(* PLC project v0.6.04_CycleSemiAuto.project, CODESYS CODESYS V3.5 SP19 Patch 1 *)
(* stored: creationDateTime 2026-08-15T14:41:18.168777, modificationDateTime 2026-08-15T14:41:18.168777 *)

(* values of E_Mode: DISABLE: Mode Désactivé / Veille de sécurité (sorties bloquées); MAINT_N1: Manuel Niveau 1 : Pilotage unitaire avec toutes sécurités actives; MAINT_N2: Manuel Niveau 2 : Pilotage dégradé (droits étendus + bypasses autorisés); SEMI_AUTO: Mode Semi-Automatique (séquenceur automatique) *)

{attribute 'qualified_only'}
{attribute 'strict'}
TYPE E_Mode : (DISABLE := 0, MAINT_N1 := 1, MAINT_N2 := 2, SEMI_AUTO := 3);
END_TYPE

(* ═══════════════════════════════════════════════════════════════ 📡 ST_Diag_Device — Structure diagnostic d'un esclave ou bus ═══════════════════════════════════════════════════════════════ *)
TYPE ST_Diag_Device : STRUCT
  Online : BOOL;  (* Esclave visible sur le bus *)
  Operational : BOOL;  (* Esclave en mode OP (opérationnel) *)
  Error : BOOL;  (* Signal de défaut actif pour cet esclave *)
  ErrorId : WORD;  (* Code défaut détaillé *)
  State : E_Diag_State;  (* Phase courante du cycle de diagnostic *)
  StateAtError : E_Diag_State;  (* Instantané de la phase lors de l'anomalie *)
END_STRUCT;
END_TYPE

(* ═══════════════════════════════════════════════════════════════ 🕹️ ST_Joystick_AxisCmd — Consigne d'axe normalisée (sortie FB_Joystick) ─────────────────────────────────────────────────────────────── 📄 Doc métier : DOC/AF/AF_Partie-08_Fonction_Joystick_v2.0.md DOC/AF/AF_Partie-03_Contrats_Composants_v2.1.md 🎯 4 champs exactement : - Enable : Autorisation globale du pipeline - StartStop : RAMPE (TRUE = accélération, FALSE = décélération normale) - SpeedRef : Consigne vitesse signée (-100.0 .. +100.0 %) - Direction : Sens d'axe (-1 = Rev, 0 = Neutre, +1 = Fwd) ═══════════════════════════════════════════════════════════════ *)
TYPE ST_Joystick_AxisCmd : STRUCT
  Enable : BOOL;  (* Autorisation FB (FALSE = neutralisation, sorties coupées) *)
  StartStop : BOOL;  (* TRUE = rampe accélération, FALSE = rampe décélération normale *)
  SpeedRef : REAL;  (* Consigne vitesse SIGNÉE -100..+100 % (signe = sens, cohérent avec Direction) *)
  Direction : INT;  (* -1 = Rev, 0 = Neutre, +1 = Fwd *)
END_STRUCT;
END_TYPE

(* values of E_Diag_State: DISABLED: Désactivé (surveillance non active); READY: Opérationnel réel, pas de défaut; INIT: Initialisation / Recherche de réseau; MONITORING: Surveillance active (états transitoires); ERROR: Anomalie de communication; SIMULATED: Bypass simulation ou bypass réseau IHM — pas le bus réel *)

{attribute 'qualified_only'}
{attribute 'strict'}
TYPE E_Diag_State : (DISABLED := 0, READY := 1, INIT := 2, MONITORING := 3, ERROR := 4, SIMULATED := 5);
END_TYPE

(* ═══════════════════════════════════════════════════════════════ 🕹️ FB_Joystick — Acquisition & traitement Hall (Homme-mort ISO 13850) ─────────────────────────────────────────────────────────────── 📄 Doc métier : DOC/AF/AF_Partie-08_Fonction_Joystick_v2.0.md DOC/AF/AF_Partie-03_Contrats_Composants_v2.1.md 🎯 Rôle : Acquisition 2 axes Hall + bouton homme-mort normatif. Pipeline par axe : FB_AxisScale → FB_Filter_PT1 → Homme-Mort → ST_Joystick_AxisCmd. Les rampes d'accélération/décélération sont gérées exclusivement par les FB de mouvement aval (FB_Winch, FB_Translation), hors de ce bloc. 🔒 Bouton homme-mort : - Armement au neutre strict (ScaleX/Y.OutPct = 0.0). - Consentement au démarrage : mouvement libre SANS surveillance du bouton (défaut, DeadmanReconfEnable := FALSE). Optionnel : reconfirmation périodique en mouvement (délai DeadmanRearmTimeout) si DeadmanReconfEnable := TRUE. - Désarmement sur maintien au neutre (durée NeutralHoldTime) + gate/mode/fin benne. 📤 Produit AxisCmdX, AxisCmdY, et signaux de diagnostic/miroir. ═══════════════════════════════════════════════════════════════ === DECLARATION (à coller dans la partie déclaration du POU FB_Joystick) === *)
FUNCTION_BLOCK FB_Joystick
  VAR_INPUT
    Enable : BOOL;  (* Active la logique *)
    Reset : BOOL;  (* Acquittement défaut *)
    PowerContactorEngaged : BOOL;  (* Conditions globales OK (chaîne AU réarmée) *)
    Mode : E_Mode;  (* Changement de mode désarme le homme-mort *)
    BenneBusy : BOOL;  (* Fin de cycle benne (front descendant) désarme le homme-mort *)
    PreserveArmingAfterBucket : BOOL;  (* TRUE uniquement pendant fermeture ExtractionSequence : enchaînement palier 1 autorisé *)
    BusCanOpenOP : ST_Diag_Device;  (* État présence nœud CAN *)
    JoystickOP : ST_Diag_Device;  (* Mode esclave CANopen actif *)
    RawX : INT;  (* Valeur brute axe X *)
    RawY : INT;  (* Valeur brute axe Y *)
    RawButton : BOOL;  (* État brut bouton *)
    BtnCalibrate : BOOL;  (* Demande de recalage neutre *)
    InvertX : BOOL := FALSE;
    InvertY : BOOL := FALSE;
    DeadbandRaw : INT := 300;  (* Zone morte en points ADC bruts (0..10000) *)
    FilterTime : TIME := TIME#0ms;  (* Filtrage premier ordre axe *)
    NeutralHoldTime : TIME := TIME#100MS;  (* Maintien continu au neutre avant désarmement *)
    DeadmanArmHoldTime : TIME := TIME#100MS;  (* Appui continu bouton requis pour armer *)
    DeadmanArmGraceTime : TIME := TIME#3S;  (* Délai de grâce post-armement avant application du désarmement neutre *)
  END_VAR
  VAR_OUTPUT
    Ready : BOOL;  (* Prêt à commuter *)
    Busy : BOOL;  (* Traitement en cours *)
    Done : BOOL;  (* Données valides dispo *)
    Error : BOOL;  (* Présence anomalie *)
    ErrorId : WORD;  (* bit0: "Échec calibration Joystick" - Valeurs RawX/Y hors plage lors du recalage *)
    AxisCmdX : ST_Joystick_AxisCmd;  (* Sortie normalisée X *)
    AxisCmdY : ST_Joystick_AxisCmd;  (* Sortie normalisée Y *)
    Button : BOOL;  (* Bouton filtré *)
    NeutralXAct : INT;  (* Point neutre X actuel pour IHM/Test *)
    NeutralYAct : INT;  (* Point neutre Y actuel pour IHM/Test *)
    SpeedXPct : REAL;  (* 🆕 Miroirs directs (maintenance) — mêmes valeurs que AxisCmdX/Y.SpeedRef/.Direction, exposés à plat pour lecture immédiate en vue instance CODESYS (pas de dépliage struct). Consigne vitesse axe X en % SIGNÉE (-100..+100), miroir AxisCmdX.SpeedRef *)
    DirectionX : INT;  (* Sens axe X (-1=Rev/0=Neutre/+1=Fwd), miroir AxisCmdX.Direction *)
    SpeedYPct : REAL;  (* Consigne vitesse axe Y en % SIGNÉE (-100..+100), miroir AxisCmdY.SpeedRef *)
    DirectionY : INT;  (* Sens axe Y (-1=Rev/0=Neutre/+1=Fwd), miroir AxisCmdY.Direction *)
    DeadmanArmed : BOOL;  (* 🆕 Geste armé (bouton appuyé au neutre) — IHM/diagnostic *)
    AtNeutral : BOOL;  (* 🆕 2026-08-07 : TRUE si les 2 axes sont en zone morte (position centrale) — IHM/diagnostic *)
  END_VAR
  VAR_IN_OUT
    NeutralXMem : INT;  (* Point neutre X persistant global *)
    NeutralYMem : INT;  (* Point neutre Y persistant global *)
  END_VAR
  VAR
    CycleTimeCalc : FB_CycleTime;
    ScaleX : FB_AxisScale;
    ScaleY : FB_AxisScale;
    FilterX : FB_Filter_PT1;
    FilterY : FB_Filter_PT1;
    CmdXVal : REAL;
    CmdYVal : REAL;
    LastCalibrate : BOOL;
    ResetEdge : R_TRIG;
    DeadmanEdge : R_TRIG;
    NeutralHoldTimer : TON;
    DeadmanArmTimer : TON;
    DeadmanArmPending : BOOL;
    DeadmanArmGraceTimer : TON;
    LastMode : E_Mode;
    BenneBusyFallEdge : F_TRIG;
  END_VAR

            

// === IMPLEMENTATION (à coller dans le corps ST du POU FB_Joystick) ===

{region "§1 Gate securite"}
// 🛑 1. GATE (Sécurités et coupures prioritaires)
IF NOT Enable OR NOT PowerContactorEngaged OR NOT BusCanOpenOP.Operational OR NOT JoystickOP.Operational THEN
    Ready := FALSE; Busy := FALSE; Done := FALSE;
    AxisCmdX.Enable := FALSE; AxisCmdX.StartStop := FALSE; AxisCmdX.SpeedRef := 0.0; AxisCmdX.Direction := 0;
    AxisCmdY.Enable := FALSE; AxisCmdY.StartStop := FALSE; AxisCmdY.SpeedRef := 0.0; AxisCmdY.Direction := 0;
    SpeedXPct := 0.0; DirectionX := 0;
    SpeedYPct := 0.0; DirectionY := 0;
    Button := FALSE;
    AtNeutral := TRUE;
    DeadmanArmed := FALSE;
    DeadmanArmPending := FALSE;
    NeutralHoldTimer(IN := FALSE, PT := NeutralHoldTime);
    DeadmanArmTimer(IN := FALSE, PT := DeadmanArmHoldTime);
    DeadmanArmGraceTimer(IN := FALSE, PT := DeadmanArmGraceTime);
    NeutralXAct := NeutralXMem;
    NeutralYAct := NeutralYMem;
    LastMode := Mode;   // 🆕 REX 2026-07-08 — pas de faux changement détecté à la réactivation
    RETURN;
END_IF;

Ready := TRUE; Busy := TRUE;

{endregion}

{region "§2 Reset acquisition timing et bouton"}
// 🔑 2. RESET DÉFAUT (front + cause disparue, Partie3 §5)
ResetEdge(CLK := Reset);
IF ResetEdge.Q AND (RawX >= 2000 AND RawX <= 8000 AND RawY >= 2000 AND RawY <= 8000) THEN
    ErrorId := ErrorId AND 16#FFFE;
END_IF;

// 📥 3. ACQUISITION TIMING & BOUTON
CycleTimeCalc();
Button := RawButton;

{endregion}

{region "§3 Calibration et mise a echelle"}
// 🎯 4. CALIBRATION DYNAMIQUE (Zone RETAIN)
IF BtnCalibrate AND NOT LastCalibrate THEN
    IF RawX >= 2000 AND RawX <= 8000 AND RawY >= 2000 AND RawY <= 8000 THEN
        NeutralXMem := RawX;
        NeutralYMem := RawY;
    ELSE
        // Un seul bit pour une seule cause (Partie3 §3)
        ErrorId := ErrorId OR 16#0001;
    END_IF;
END_IF;
Error := (ErrorId <> 16#0000);
LastCalibrate := BtnCalibrate;

// 🧮 4bis. MISE À L'ÉCHELLE (avant homme-mort — le neutre s'évalue sur les 2 axes déjà deadbandés)
ScaleX(RawIn := RawX, Neutral := NeutralXMem, DeadbandRaw := DeadbandRaw);
ScaleY(RawIn := RawY, Neutral := NeutralYMem, DeadbandRaw := DeadbandRaw);
AtNeutral := (ScaleX.OutPct = 0.0) AND (ScaleY.OutPct = 0.0);   // 🆕 2026-08-07 : IHM/diagnostic — position centrale (zone morte)

{endregion}

{region "§4 Desarmements changement mode et fin benne"}
// 4ter-bis. CHANGEMENT DE MODE : désarme le homme-mort dès que Mode change
// (MAINT_N1/N2/SEMI_AUTO/AUTO). Évite qu'une commande en cours traverse le changement
// de mode et soit réinterprétée soudainement. Repassage par le neutre + nouvel appui exigé.
IF Mode <> LastMode THEN
    DeadmanArmed := FALSE;
    DeadmanArmPending := FALSE;   // 🆕 2026-08-07 — nouvel appui exigé après changement de mode
END_IF;
LastMode := Mode;

// 4ter-ter. FIN DE CYCLE BENNE : désarmement général pour qu'une fermeture manuelle
// ne démarre jamais M1/M2 par surprise. Exception : ExtractionSequence garde l'armement
// pendant sa fermeture (enchaînement palier 1 sous ses propres interlocks synchro/position).
BenneBusyFallEdge(CLK := BenneBusy);
IF BenneBusyFallEdge.Q AND NOT PreserveArmingAfterBucket THEN
    DeadmanArmed := FALSE;
    DeadmanArmPending := FALSE;   // 🆕 2026-08-07 — nouvel appui exigé après fin de cycle benne
END_IF;

{endregion}

{region "§5 Armement homme mort"}
// 4ter. BOUTON HOMME-MORT — armement par MAINTIEN (DeadmanArmHoldTime), indépendant de la
// position des axes pendant l'appui.
// 🔧 2026-08-07 (retour terrain) : l'ancien armement ("front bouton" ET "axes strictement à
// 0.0 sur le MÊME scan") échouait dès que l'opérateur poussait le joystick quelques ms après
// avoir appuyé — trop contraignant en pratique (le geste naturel "j'appuie PUIS je pousse" ratait
// systématiquement la fenêtre d'un seul scan). Nouvelle séquence : appui (front) → maintien
// DeadmanArmHoldTime (100 ms) → armé, quelle que soit la position des axes durant ce maintien.
// Relâchement AVANT la fin du maintien = tentative annulée (DeadmanArmPending retombe), un
// nouvel appui (front) est requis — pas d'armement différé "surprise" sur un appui prolongé après
// un désarmement (mode/benne/neutre). Sûr même si le joystick est déjà hors zone morte à la fin
// du maintien : les rampes d'accel/décel restent gérées par les FB aval (FB_Winch/FB_Translation,
// cf. §"Rôle" en tête de fichier), donc pas de démarrage brutal possible côté ce FB.
DeadmanEdge(CLK := RawButton);
IF DeadmanEdge.Q THEN
    DeadmanArmPending := TRUE;
END_IF;
IF NOT RawButton THEN
    DeadmanArmPending := FALSE;
END_IF;

// 🛡️ SÉCURITÉ C4 (ISO 13849) : armement STRICTEMENT conditionné par DeadmanArmPending.
// Tout désarmement (changement de mode, fin de cycle benne, passage neutre prolongé)
// efface DeadmanArmPending et EXIGE un nouvel appui conscient (front montant de RawButton).
DeadmanArmTimer(IN := DeadmanArmPending AND NOT DeadmanArmed, PT := DeadmanArmHoldTime);
IF DeadmanArmTimer.Q THEN
    DeadmanArmed := TRUE;
    DeadmanArmPending := FALSE;
END_IF;

// ⏱️ 4bis. GESTION DU DÉSARMEMENT PAR MAINTIEN AU NEUTRE
DeadmanArmGraceTimer(IN := DeadmanArmed, PT := DeadmanArmGraceTime);
NeutralHoldTimer(IN := DeadmanArmed AND AtNeutral AND DeadmanArmGraceTimer.Q,
                 PT := NeutralHoldTime);
IF NeutralHoldTimer.Q THEN
    DeadmanArmed := FALSE;      // Neutre maintenu après la grâce = désarmement
END_IF;

{endregion}

{region "§6 Pipeline axe X"}
// 🕹️ 5. PIPELINE TRAITEMENT — AXE X
IF InvertX THEN
    FilterX(ValueIn := -ScaleX.OutPct, TimeConst := FilterTime, CycleTimeS := CycleTimeCalc.CycleTimeS);
ELSE
    FilterX(ValueIn := ScaleX.OutPct, TimeConst := FilterTime, CycleTimeS := CycleTimeCalc.CycleTimeS);
END_IF;

// Consigne forcée à 0.0 tant que le geste n'est pas armé (homme-mort)
CmdXVal := SEL(DeadmanArmed, 0.0, FilterX.ValueOut);

// Mapping Sortie Standardisée Axe X
AxisCmdX.Enable := TRUE;
AxisCmdX.SpeedRef := CmdXVal;
AxisCmdX.StartStop := (ABS(CmdXVal) > 0.1);

IF CmdXVal > 0.1 THEN
    AxisCmdX.Direction := 1;
ELSIF CmdXVal < -0.1 THEN
    AxisCmdX.Direction := -1;
ELSE
    AxisCmdX.Direction := 0;
    AxisCmdX.SpeedRef := 0.0;
END_IF;

// Miroirs maintenance
SpeedXPct := AxisCmdX.SpeedRef;
DirectionX := AxisCmdX.Direction;

{endregion}

{region "§7 Pipeline axe Y et sorties"}
// 🕹️ 6. PIPELINE TRAITEMENT — AXE Y
IF InvertY THEN
    FilterY(ValueIn := -ScaleY.OutPct, TimeConst := FilterTime, CycleTimeS := CycleTimeCalc.CycleTimeS);
ELSE
    FilterY(ValueIn := ScaleY.OutPct, TimeConst := FilterTime, CycleTimeS := CycleTimeCalc.CycleTimeS);
END_IF;

// Consigne forcée à 0.0 tant que le geste n'est pas armé (homme-mort)
CmdYVal := SEL(DeadmanArmed, 0.0, FilterY.ValueOut);

// Mapping Sortie Standardisée Axe Y
AxisCmdY.Enable := TRUE;
AxisCmdY.SpeedRef := CmdYVal;
AxisCmdY.StartStop := (ABS(CmdYVal) > 0.1);

IF CmdYVal > 0.1 THEN
    AxisCmdY.Direction := 1;
ELSIF CmdYVal < -0.1 THEN
    AxisCmdY.Direction := -1;
ELSE
    AxisCmdY.Direction := 0;
    AxisCmdY.SpeedRef := 0.0;
END_IF;

// Miroirs maintenance
SpeedYPct := AxisCmdY.SpeedRef;
DirectionY := AxisCmdY.Direction;

// 📤 7. VALIDATION DES SORTIES ÉTAT
NeutralXAct := NeutralXMem;
NeutralYAct := NeutralYMem;
Done := NOT Error;

{endregion}

          
END_FUNCTION_BLOCK

(* ═══════════════════════════════════════════════════════════════ 📐 FB_AxisScale — Mise à l'échelle d'un axe joystick Hall ─────────────────────────────────────────────────────────────── 📄 Extrait depuis le projet CODESYS (Device.export, JOYSTICK/) 🎯 Normalise une valeur brute (0..10000) par rapport au neutre calibré et applique une zone morte en unités brutes (compte ADC, pas en %). Sortie : OutPct ∈ [-100.0 .. +100.0] (0.0 si dans la deadband) 🔧 2026-08-07 (demande client) : Deadband (REAL, %) → DeadbandRaw (INT, compte brut 0..10000). Raison : plus simple à régler directement depuis le bruit mesuré au neutre (ex: ±200 sur le terrain → DeadbandRaw=300 avec marge), sans recalculer un % à chaque calibration. ═══════════════════════════════════════════════════════════════ 📄 Docs : DOC/AF/AF_Partie-08_Fonction_Joystick_v2.0.md *)
FUNCTION_BLOCK FB_AxisScale
  VAR_INPUT
    RawIn : INT;  (* / Valeur brute (0..10000) *)
    Neutral : INT;  (* / Point milieu calibré *)
    DeadbandRaw : INT;  (* / Zone morte en unités brutes (compte ADC, ex: 300 sur plage 0..10000) *)
  END_VAR
  VAR_OUTPUT
    OutPct : REAL;  (* / Valeur finale (-100.0..100.0) *)
  END_VAR
  VAR
    Delta : REAL;
  END_VAR

            

IF RawIn >= Neutral THEN
    Delta := INT_TO_REAL(10000 - Neutral);
    IF Delta > 0.0 THEN
        OutPct := (INT_TO_REAL(RawIn - Neutral) / Delta) * 100.0;
    ELSE
        OutPct := 0.0;
    END_IF;
ELSE
    Delta := INT_TO_REAL(Neutral);
    IF Delta > 0.0 THEN
        OutPct := (INT_TO_REAL(RawIn - Neutral) / Delta) * 100.0;
    ELSE
        OutPct := 0.0;
    END_IF;
END_IF;

IF ABS(RawIn - Neutral) <= DeadbandRaw THEN
    OutPct := 0.0;
END_IF;

// 🛡️ Limitation de plage : une valeur brute hors plage nominale ne doit jamais
// produire une consigne supérieure à ±100 %. Ce garde-fou protège les
// consommateurs en aval, notamment la translation M3.
OutPct := LIMIT(-100.0, OutPct, 100.0);

          
END_FUNCTION_BLOCK

(* ═══════════════════════════════════════════════════════════════ ⏱️ FB_CycleTime — Mesure du temps de cycle réel de la tâche ─────────────────────────────────────────────────────────────── 📄 Doc métier : DOC/AF/AF_Partie-08_Fonction_Joystick_v2.0.md §2 (base de temps utilisée par FB_Filter_PT1, composé dans FB_Joystick) ═══════════════════════════════════════════════════════════════ *)
FUNCTION_BLOCK FB_CycleTime
  VAR_INPUT
    DefaultValueS : REAL := 0.004;  (* Valeur de secours par défaut (ex. 4ms) *)
  END_VAR
  VAR_OUTPUT
    CycleTimeS : REAL;  (* Temps écoulé réel calculé (secondes) *)
  END_VAR
  VAR
    TimeCurrent : TIME;  (* Temps système actuel *)
    TimeLast : TIME;  (* Empreinte de temps du cycle précédent *)
    DeltaTimeMs : UDINT;  (* Écart brut calculé (ms) *)
    InitDone : BOOL;  (* Drapeau d'initialisation du premier cycle *)
  END_VAR

            

// 1. ACQUISITION DU TEMPS SYSTÈME
TimeCurrent := TIME();

// 2. INITIALISATION UNIQUE AU PREMIER CYCLE
IF NOT InitDone THEN
    TimeLast := TimeCurrent;
    InitDone := TRUE;
    CycleTimeS := DefaultValueS;
    RETURN;
END_IF;

// 3. CALCUL DU DELTA EN MILLISECONDES
DeltaTimeMs := TIME_TO_UDINT(TimeCurrent - TimeLast);

// 4. CONVERSION ET CHARGE DE SECOURS
IF DeltaTimeMs > 0 THEN
    CycleTimeS := UDINT_TO_REAL(DeltaTimeMs) / 1000.0;
ELSE
    CycleTimeS := DefaultValueS;
END_IF;

// 5. ARCHIVAGE POUR LE PROCHAIN CYCLE
TimeLast := TimeCurrent;

          
END_FUNCTION_BLOCK

(* ═══════════════════════════════════════════════════════════════ 🔁 FB_Filter_PT1 — Filtre passe-bas premier ordre (PT1 numérique) ─────────────────────────────────────────────────────────────── 📄 Extrait depuis le projet CODESYS (Device.export, JOYSTICK/) 🎯 Filtre exponentiel discret : y[k] = α·x[k] + (1-α)·y[k-1] où α = CycleTimeS / (T + CycleTimeS), T = TimeConst en secondes. ⚠️ Si TimeConst = 0 ou CycleTimeS = 0, sortie = entrée (pass-through). ═══════════════════════════════════════════════════════════════ 📄 Docs : DOC/AF/AF_Partie-08_Fonction_Joystick_v2.0.md *)
FUNCTION_BLOCK FB_Filter_PT1
  VAR_INPUT
    ValueIn : REAL;  (* / Consigne brute entrée *)
    TimeConst : TIME;  (* / Constante de temps du filtre *)
    CycleTimeS : REAL;  (* / Temps de cycle réel en secondes *)
  END_VAR
  VAR_OUTPUT
    ValueOut : REAL;  (* / Consigne filtrée sortie *)
  END_VAR
  VAR
    T : REAL;
    Alpha : REAL;
  END_VAR

            

T := TIME_TO_REAL(TimeConst) / 1000.0; // ms → s

IF T <= 0.0 OR CycleTimeS <= 0.0 THEN
    ValueOut := ValueIn;
ELSE
    Alpha    := CycleTimeS / (T + CycleTimeS);
    ValueOut := Alpha * ValueIn + (1.0 - Alpha) * ValueOut;
END_IF;

          
END_FUNCTION_BLOCK
